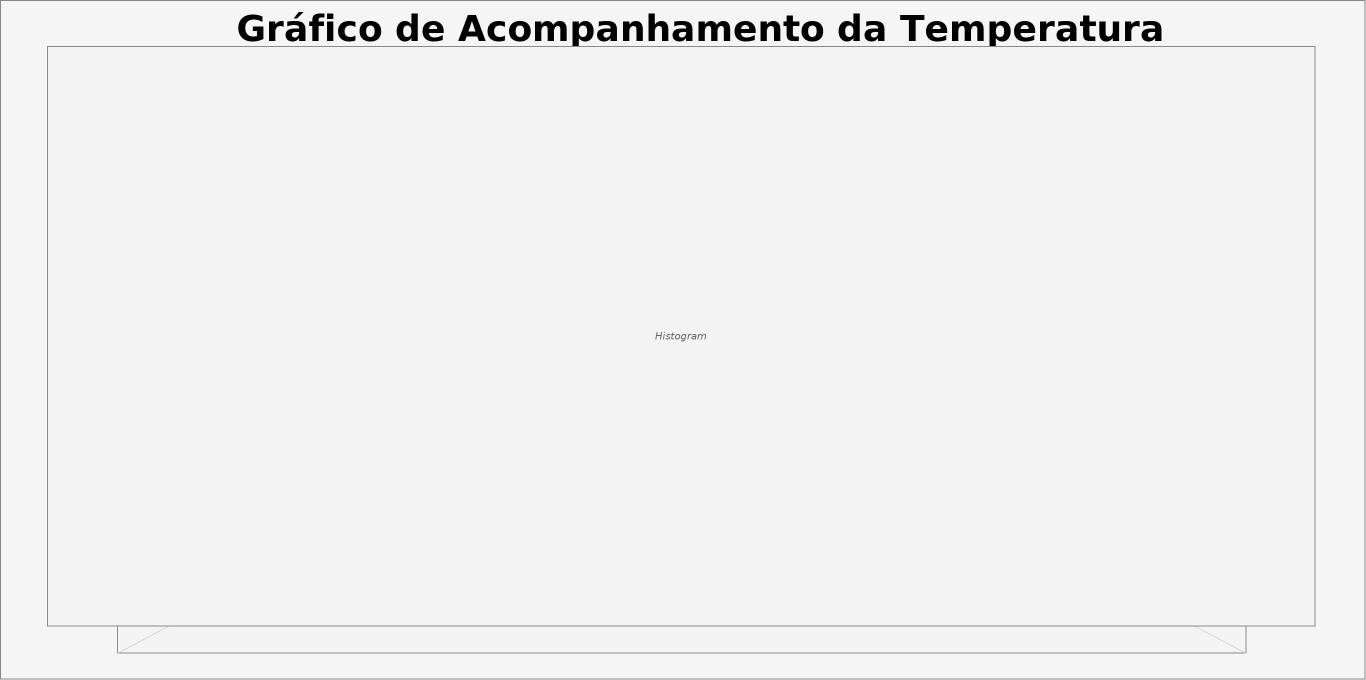
VISUALIZATION Grafico_3  // 1366x680
    Image (117,53 1129x600), image: ImagePool.teseagraf
    Histogram (47,46 1268x580), scale format: %.1f, scale 0..150
        p1518820177: GVL_P.arrTempVisu021
        p102497268: GVL_P.arrTempVisu021
        p788070771: ARRAY [1..720] OF REAL
    Label (262,7 877x43), "Gráfico de Acompanhamento da Temperatura"
    Histogram (47,46 1268x580), scale format: %.1f, scale 0..150
        p1518820177: GVL_P.arrTemp021
        p102497268: GVL_P.arrTemp021
        p788070771: ARRAY [1..720] OF REAL
END_VISUALIZATION

(* stored: Version 1.1.0.1, ProductVersion 3.1.4024.12
   Visu Grafico_3: Id {f92ea68b-f5cb-4711-a133-7b1efca3553b} *)
